{attribute addProperty BoxType "EL4021-0000-0016"}
{attribute addProperty Id "AO_OutputsAT %Q*AO_Outputs_F57FA4F91620WcStateAT %I*WcState_28A8677510.1250InfoDataAT %I*InfoData_BC63D37F80100"}
{attribute addProperty CRC "1097990690"}
{attribute addProperty SizeInBites "97"}
{attribute addProperty SizeInBytes "12.125"}
TYPE EL4021_50B5189C :
STRUCT
	{attribute addProperty Name "AO_Outputs"}
	AO_Outputs : AO_Outputs_F57FA4F9;
	{attribute addProperty Name "WcState"}
	WcState : WcState_28A86775;
	{attribute addProperty Name "InfoData"}
	InfoData : InfoData_BC63D37F;
END_STRUCT
END_TYPE

(* stored: Version 1.2.0.0, ProductVersion 3.1.4024.9
   DUT EL4021_50B5189C: Id {9c93034f-59aa-458d-a73b-8bce4f920704} *)
